SUBAPPLICATION Uebung_028_AX (* Analog-Eingang *)
  (* Standard: 61499-2; Description: Copyright (c) 2023 Meisterschulen am Ostbahnhof This program and the accompanying materials are made available under the terms of the Eclipse Public License 2.0 which is available at https://www.eclipse.org/legal/epl-2.0/ SPDX-License-Identifier: EPL-2.0 *)
  (* Version 1.0, 2023-10-23, Franz Höpfinger, Meisterschulen am Ostbahnhof, initial API and implementation and/or initial documentation *)
  PACKAGE Uebungen;
  IMPORT logiBUS::io::DI::logiBUS_DI::Input_I1;
  IMPORT logiBUS::io::DQ::logiBUS_DO::Output_Q1;
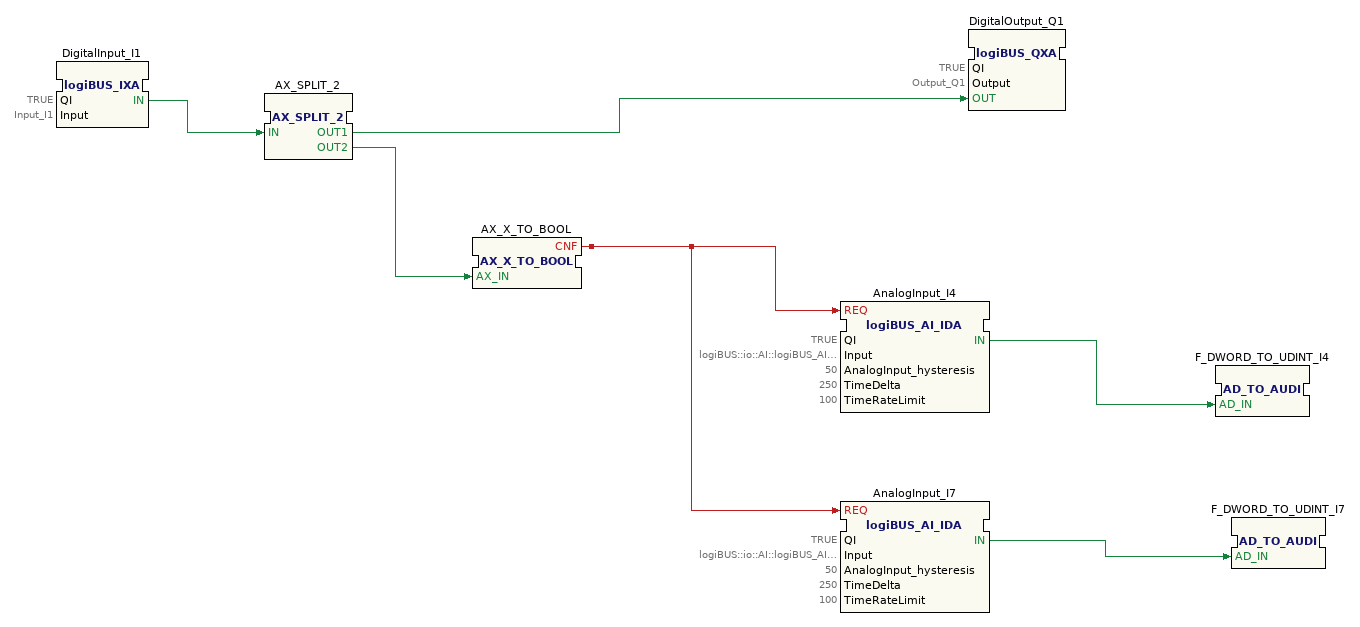
  FBS
    DigitalOutput_Q1 : logiBUS::io::DQ::logiBUS_QXA(QI := TRUE, Output := Output_Q1);
    DigitalInput_I1 : logiBUS::io::DI::logiBUS_IXA(QI := TRUE, Input := Input_I1);
    AnalogInput_I4 : logiBUS::io::AI::logiBUS_AI_IDA(QI := TRUE, Input := logiBUS::io::AI::logiBUS_AI::AnalogInput_I4, AnalogInput_hysteresis := 50, TimeDelta := 250, TimeRateLimit := 100);
    AnalogInput_I7 : logiBUS::io::AI::logiBUS_AI_IDA(QI := TRUE, Input := logiBUS::io::AI::logiBUS_AI::AnalogInput_I7, AnalogInput_hysteresis := 50, TimeDelta := 250, TimeRateLimit := 100);
    F_DWORD_TO_UDINT_I7 : adapter::conversion::unidirectional::AD_TO_AUDI;
    F_DWORD_TO_UDINT_I4 : adapter::conversion::unidirectional::AD_TO_AUDI;
    AX_X_TO_BOOL : adapter::conversion::unidirectional::AX_X_TO_BOOL;
    AX_SPLIT_2 : adapter::events::unidirectional::AX_SPLIT_2;
  END_FBS
  EVENT_CONNECTIONS
    AX_X_TO_BOOL.CNF TO AnalogInput_I4.REQ;
    AX_X_TO_BOOL.CNF TO AnalogInput_I7.REQ;
  END_CONNECTIONS
  ADAPTER_CONNECTIONS
    AnalogInput_I7.IN TO F_DWORD_TO_UDINT_I7.AD_IN;
    AX_SPLIT_2.OUT1 TO DigitalOutput_Q1.OUT;
    AnalogInput_I4.IN TO F_DWORD_TO_UDINT_I4.AD_IN;
    DigitalInput_I1.IN TO AX_SPLIT_2.IN;
    AX_SPLIT_2.OUT2 TO AX_X_TO_BOOL.AX_IN;
  END_CONNECTIONS
END_SUBAPPLICATION
